Staubli VAL3: Deb2304.dtx

dio dPowerlinkSorti = {link=POWERLINK-1\%Q0}
mdesc mNomSpeed
mdesc mlent = {accel=9, vel=30, decel=9, blend=off}
tool tstylo = {z=100, fatherId=flange[0], ioLink=valve1}
jointRx ja[5]
  [0] = {j1=-141.592538, j2=84.02454, j3=39.666751, j4=0.388019, j5=55.73836, j6=91.723919}
  [1] = {j1=-141.797065, j2=55.548957, j3=26.304021, j4=0.325386, j5=97.577607, j6=91.780733}
  [2] = {j1=-1.061441, j2=69.857939, j3=0.585564, j4=-0.646318, j5=109.792733, j6=232.256985}
  [3] = {j1=-1.782017, j2=63.511465, j3=34.980386, j4=-0.618292, j5=81.739303, j6=231.843932}
  [4] = {j1=-1.782031, j2=69.640192, j3=39.18089, j4=-0.645507, j5=71.410438, j6=231.960844}
num nPowerlink
public dio diECAT1_0 = {link=POWERLINK-1\%I0}
public dio diECAT1_1 = {link=POWERLINK-1\%I1}
public dio diECAT1_2 = {link=POWERLINK-1\%I2}
public dio diECAT1_3 = {link=POWERLINK-1\%I3}
public dio diECAT1_4 = {link=POWERLINK-1\%I4}
public dio diECAT1_5 = {link=POWERLINK-1\%I5}
public dio diECAT1_6 = {link=POWERLINK-1\%I6}
public dio diECAT1_7 = {link=POWERLINK-1\%I7}
public dio diECAT1_8 = {link=POWERLINK-1\%I8}
public dio diECAT1_9 = {link=POWERLINK-1\%I9}
public dio diECAT1_10 = {link=POWERLINK-1\%I10}
public dio diECAT1_11 = {link=POWERLINK-1\%I11}
public dio diECAT1_12 = {link=POWERLINK-1\%I12}
public dio diECAT1_13 = {link=POWERLINK-1\%I13}
public dio diECAT1_14 = {link=POWERLINK-1\%I14}
public dio diECAT1_15 = {link=POWERLINK-1\%I15}
public dio diECAT1_16 = {link=POWERLINK-1\%I16}
public dio doECAT1_0 = {link=POWERLINK-1\%Q0}
public dio doECAT1_1 = {link=POWERLINK-1\%Q1}
bool x[8]
bool rbt_ready
num co_x
num co_y
bool y[8]
